FUNCTION_BLOCK TLController_Centralised (* Composite Function Block Type *)
  (* Standard: 61499-2 *)
  (* Version 0.2, 2003-12-05, JHC, Rockwell Automation, Renamed from NEWCOMPFB. *)
  (* Version 0.1, 2002-01-08, JHC, Rockwell Automation, Added DLY FB as example. *)
  (* Version 0.0, 2000-05-27, JHC, Rockwell Automation *)
  (* Compiler header: package fb.rt.template; *)
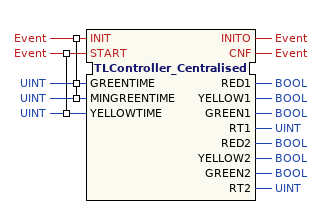
  EVENT_INPUT
    INIT WITH GREENTIME, MINGREENTIME; (* Initialization Request *)
    START WITH YELLOWTIME;
  END_EVENT
  EVENT_OUTPUT
    INITO; (* Initialization Confirm *)
    CNF;
  END_EVENT
  VAR_INPUT
    GREENTIME : UINT;
    MINGREENTIME : UINT;
    YELLOWTIME : UINT;
  END_VAR
  VAR_OUTPUT
    RED1 : BOOL;
    YELLOW1 : BOOL;
    GREEN1 : BOOL;
    RT1 : UINT;
    RED2 : BOOL;
    YELLOW2 : BOOL;
    GREEN2 : BOOL;
    RT2 : UINT;
  END_VAR
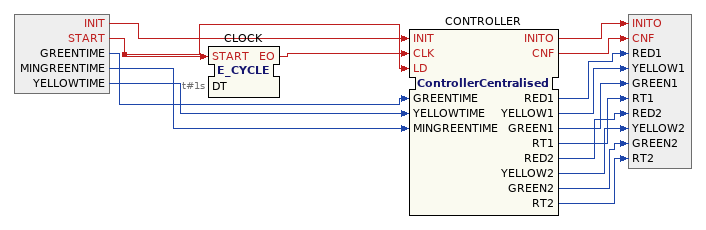
  FBS
    CLOCK : E_CYCLE(DT := t#1s);
    CONTROLLER : ControllerCentralised;
  END_FBS
  EVENT_CONNECTIONS
    START TO CLOCK.START;
    CLOCK.EO TO CONTROLLER.CLK;
    INIT TO CONTROLLER.INIT;
    START TO CONTROLLER.LD;
    CONTROLLER.INITO TO INITO;
    CONTROLLER.CNF TO CNF;
  END_CONNECTIONS
  DATA_CONNECTIONS
    GREENTIME TO CONTROLLER.GREENTIME;
    MINGREENTIME TO CONTROLLER.MINGREENTIME;
    YELLOWTIME TO CONTROLLER.YELLOWTIME;
    CONTROLLER.RED1 TO RED1;
    CONTROLLER.YELLOW1 TO YELLOW1;
    CONTROLLER.GREEN1 TO GREEN1;
    CONTROLLER.RT1 TO RT1;
    CONTROLLER.RT2 TO RT2;
    CONTROLLER.GREEN2 TO GREEN2;
    CONTROLLER.YELLOW2 TO YELLOW2;
    CONTROLLER.RED2 TO RED2;
  END_CONNECTIONS
END_FUNCTION_BLOCK
